Universal Robots PolyScope program: P1Artemjoan.urp

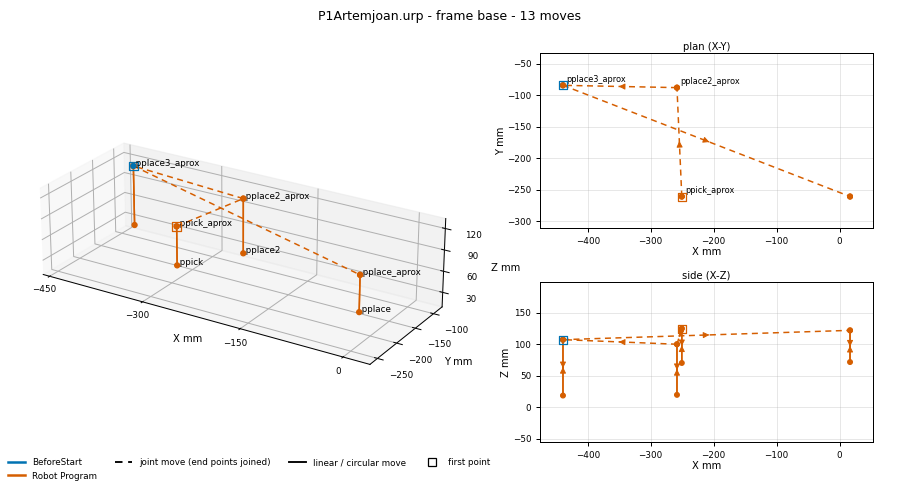
[picture p0: tool path of P1Artemjoan.urp in frame base, 13 of 14 moves have a stored position in this frame; points joined in program order, loops and branches not executed]
Program P1Artemjoan (installation=default directory=/programs createdIn=5.13.0 lastSavedIn=5.13.0 robotSerialNumber=20195300809)
Calibrated DH parameters: a=[-0.000085, -0.20076, -0.212369, 0.000121, -0.000118, 0]; d=[0.15185, -26.306375, 24.753047, 1.684739, 0.085386, 0.092088]; alpha=[1.572149, -0.00522, -0.011864, 1.571339, -1.571085, 0]; deltaTheta=[0, 0.599885, -0.513355, -0.086555, 0.000006, 0]
InitVariablesNode variables(variable(name=cont, expression=0))
BeforeStart
  URCap Gripper Activate (Robotiq_Grippers, Robotiq Inc.) dataModel(ResetAndActivateKey=false)
  MoveJ speed 60 deg/s, acceleration 80 deg/s^2 (useActiveTCP=true) feature=Base
    Waypoint relative (Relative): relativeFromPosition TCP in base x=-111.382 y=-330.88 z=200.488 mm, rx=-0.0269 ry=-3.1213 rz=0.0929 rad; joints [-85.73, -94.459, -65.933, -106.296, 88.069, 5.76] deg; TCP offset x=0 y=0 z=177.62 mm, rx=0 ry=0 rz=0 rad; TCP in base x=-111.373 y=-330.878 z=200.514 mm, rx=-0.0269 ry=-3.1214 rz=0.093 rad; joints [-85.731, -94.458, -65.928, -106.299, 88.073, 5.759] deg
  SuppressedNode
    Set DigitalOutput pin=digital_out[0]; digitalValue=1
  MoveJ speed 60 deg/s, acceleration 80 deg/s^2 (useActiveTCP=true) feature=Base
    Waypoint pplace3_aprox: TCP in base x=-439.306 y=-84.24 z=107.169 mm, rx=-2.1844 ry=2.2578 rz=0 rad; joints [-152.338, -122.258, -52.117, -95.614, 89.263, -149.991] deg
  URCap Gripper (Robotiq_Grippers, Robotiq Inc.) dataModel(position=21.56862745098039, force=0.0, speed=100.0, positionInDouble=21.56862745098039, forceInDouble=0.0, speedInDouble=100.0, slaveIds=[9], blocking=true)
Robot Program (runOnlyOnce=false)
  Folder pick
    MoveJ speed 60 deg/s, acceleration 80 deg/s^2 (useActiveTCP=true) feature=Base
      Waypoint ppick_aprox: motionParameters(blendRadius=0.02); TCP in base x=-250.628 y=-260.855 z=124.733 mm, rx=2.1844 ry=-2.2578 rz=0.0004 rad; joints [-112.874, -99.109, -79.894, -90.971, 89.386, -110.608] deg
    MoveL speed 250 mm/s, acceleration 1200 mm/s^2 (useActiveTCP=true) feature=Base
      Waypoint ppick: TCP in base x=-250.6 y=-260.834 z=70.124 mm, rx=-2.1844 ry=2.2578 rz=0 rad; joints [-112.81, -100.574, -92.939, -76.47, 89.371, -110.715] deg
      Wait DigitalInput pin=digital_in[0]; digitalValue=0
      URCap Gripper (Robotiq_Grippers, Robotiq Inc.) dataModel(position=100.0, force=0.0, speed=100.0, positionInDouble=100.0, forceInDouble=0.0, speedInDouble=100.0, slaveIds=[9], blocking=true)
      Waypoint ppick_aprox: motionParameters(blendRadius=0.02); TCP in base x=-250.628 y=-260.855 z=124.733 mm, rx=2.1844 ry=-2.2578 rz=0.0004 rad; joints [-112.874, -99.109, -79.894, -90.971, 89.386, -110.608] deg
  Folder place
    If cont≟3
      URCap Grip Check (Robotiq_Grippers, Robotiq Inc.) dataModel(ObjectDetectedKey=true, DimensionDimensionPositiveGapKey=5.0, DimensionNegativeGapKey=5.0, GripperIdKey=1, ModelDefinedKey=true, DimensionValidationKey=true, DimensionKey=50.0); state(isChildrenLocked=true)
        URCap If (Robotiq_Grippers, Robotiq Inc.)
          Popup Message (haltProgram=false message=thick piece inputType=Text)
          MoveJ speed 60 deg/s, acceleration 80 deg/s^2 (useActiveTCP=true) feature=Base
            Waypoint pplace2_aprox: motionParameters(blendRadius=0.02); TCP in base x=-258.287 y=-87.902 z=99.884 mm, rx=-2.1844 ry=2.2578 rz=0 rad; joints [-132.726, -76.109, -108.542, -85.335, 89.466, -130.602] deg
          MoveL speed 250 mm/s, acceleration 1200 mm/s^2 (useActiveTCP=true) feature=Base
            Waypoint pplace2: TCP in base x=-258.29 y=-87.9 z=19.5 mm, rx=-2.1845 ry=2.2578 rz=0 rad; joints [-132.589, -82.329, -126.469, -61.184, 89.501, -130.719] deg
            URCap Gripper (Robotiq_Grippers, Robotiq Inc.) dataModel(position=21.56862745098039, force=0.0, speed=100.0, positionInDouble=21.56862745098039, forceInDouble=0.0, speedInDouble=100.0, slaveIds=[9], blocking=true)
            Waypoint pplace2_aprox: motionParameters(blendRadius=0.02); TCP in base x=-258.287 y=-87.902 z=99.884 mm, rx=-2.1844 ry=2.2578 rz=0 rad; joints [-132.726, -76.109, -108.542, -85.335, 89.466, -130.602] deg
        URCap Else (Robotiq_Grippers, Robotiq Inc.)
          Popup Message (haltProgram=false message=thin piece inputType=Text)
          MoveJ speed 60 deg/s, acceleration 80 deg/s^2 (useActiveTCP=true) feature=Base
            Waypoint pplace3_aprox: motionParameters(blendRadius=0.02); TCP in base x=-439.306 y=-84.24 z=107.169 mm, rx=-2.1844 ry=2.2578 rz=0 rad; joints [-152.338, -122.258, -52.117, -95.614, 89.263, -149.991] deg
          MoveL speed 250 mm/s, acceleration 1200 mm/s^2 (useActiveTCP=true) feature=Base
            Waypoint pplace3: TCP in base x=-439.307 y=-84.277 z=18.402 mm, rx=-2.1845 ry=2.2577 rz=0 rad; joints [-152.291, -124.722, -72.211, -73.051, 89.255, -150.215] deg
            URCap Gripper (Robotiq_Grippers, Robotiq Inc.) dataModel(position=21.56862745098039, force=0.0, speed=100.0, positionInDouble=21.56862745098039, forceInDouble=0.0, speedInDouble=100.0, slaveIds=[9], blocking=true)
            Waypoint pplace3_aprox: motionParameters(blendRadius=0.02); TCP in base x=-439.306 y=-84.24 z=107.169 mm, rx=-2.1844 ry=2.2578 rz=0 rad; joints [-152.338, -122.258, -52.117, -95.614, 89.263, -149.991] deg
      cont := 0
    Else 
      MoveJ speed 60 deg/s, acceleration 80 deg/s^2 (useActiveTCP=true) feature=Base
        Waypoint pplace_aprox: motionParameters(blendRadius=0.02); TCP in base x=16.502 y=-260.806 z=121.927 mm, rx=-2.1845 ry=2.2577 rz=0.0001 rad; joints [-56.559, -72.739, -104.959, -92.289, 89.485, -54.369] deg
      MoveL speed 250 mm/s, acceleration 1200 mm/s^2 (useActiveTCP=true) feature=Base
        Waypoint pplace: TCP in base x=16.487 y=-260.78 z=71.591 mm, rx=2.1843 ry=-2.2578 rz=0.0001 rad; joints [-56.455, -73.794, -117.86, -78.324, 89.475, -54.418] deg
        URCap Gripper (Robotiq_Grippers, Robotiq Inc.) dataModel(position=21.56862745098039, force=0.0, speed=100.0, positionInDouble=21.56862745098039, forceInDouble=0.0, speedInDouble=100.0, slaveIds=[9], blocking=true)
        Waypoint pplace_aprox: motionParameters(blendRadius=0.02); TCP in base x=16.502 y=-260.806 z=121.927 mm, rx=-2.1845 ry=2.2577 rz=0.0001 rad; joints [-56.559, -72.739, -104.959, -92.289, 89.485, -54.369] deg
        cont := cont+1
Thread Thread_1 (runOnlyOnce=false)
  Set DigitalOutput pin=digital_out[0]; digitalValue=1
  Wait DigitalInput pin=digital_in[0]; digitalValue=0
  Set DigitalOutput pin=digital_out[0]; digitalValue=0
  Wait DigitalInput pin=digital_in[0]; digitalValue=1
